INTERFACE I_MessageData

PROPERTY DirRoot : POINTER to string(255)
SET
END_SET
END_PROPERTY

PROPERTY ErrorIndex : reference to uint
SET
END_SET
END_PROPERTY

PROPERTY FileRoot : pointer to string(255)
SET
END_SET
END_PROPERTY

PROPERTY LocalTime : pointer to DT
SET
END_SET
END_PROPERTY

PROPERTY MessageIndex : reference to uint
SET
END_SET
END_PROPERTY

PROPERTY MsgList : pointer to ARRAY[1..GVL_MSG.MAX_MESSAGE] OF st_message
SET
END_SET
END_PROPERTY

END_INTERFACE

(* stored: Version 1.1.0.1
   Itf I_MessageData: Id {1f83987b-9a61-489c-8981-74c45e72c9a1}
   Property DirRoot: Id {8950e3b3-bc38-4abf-a54a-3b099a75c492}
   Set Set: Id {3d3c4b37-6b11-4080-ae30-dc21229fb6b5}
   Property ErrorIndex: Id {3d500aac-d1bd-488d-9956-87daf56f27b7}
   Set Set: Id {3a300903-e8c4-42eb-8097-795e0c316139}
   Property FileRoot: Id {05188378-bc2a-42ff-bf06-59994d8513ce}
   Set Set: Id {cc5898ce-efe0-48ad-b884-b4dc1be08594}
   Property LocalTime: Id {075c3910-430e-4af4-ad3b-bb1ccb6bfe0d}
   Set Set: Id {d57294ba-59c8-41cf-8cf9-3f746e7e12f2}
   Property MessageIndex: Id {ddebc67c-73e9-43ea-ad28-c8233c3ce2e9}
   Set Set: Id {2e14246c-dc33-4970-8321-676d2163c3e4}
   Property MsgList: Id {cce934bd-c5e1-440c-9f14-df4c5c1500e5}
   Set Set: Id {6c4cefd8-a614-4fb1-8d9c-a46e631f9a16} *)
